FUNCTION F_SEND_EVENTLOGGER_MSG : BOOL
VAR_INPUT
	fbMessage:									TcEventEntry;
END_VAR
VAR
	bInit : 									BOOL; 
    bSend : 									BOOL; 
    fbMsg : 									FB_TcMessage; 
END_VAR

IF( fbMessage.nEventId = GVL_EventLogger.fbPrevMsg.nEventId
	AND fbMessage.eSeverity = GVL_EventLogger.fbPrevMsg.eSeverity) THEN
	bInit:=FALSE;
	bSend:=FALSE;
ELSE
	bInit:=TRUE;
	bSend:=TRUE;
END_IF

IF bInit THEN
    bInit := FALSE; 
    fbMsg.CreateEx(fbMessage, 0); 
END_IF

IF bSend THEN 
    bSend := FALSE; 
    fbMsg.Send(0); 
	GVL_EventLogger.fbPrevMsg:=fbMessage;
	GVL_EventLogger.udiPrevMsgId:=fbMessage.nEventId;
END_IF

END_FUNCTION

(* stored: Version 1.1.0.1, ProductVersion 3.1.4024.12
   POU F_SEND_EVENTLOGGER_MSG: Id {67cbd701-4cfd-4cbb-883d-7330421cfcba}, SpecialFunc None *)
